Staubli VAL3: onF6Event.pgx

program onF6Event()
  local string l_sString
  local num l_nResult
  local bool l_bUndo
  local string l_sPaste
begin
  // look if the bButton is enable
  if bButton[5]
    //
    //  Duplicate
    //
    l_sPaste=sEvent
    call alreadyExist(l_sPaste,l_bUndo)
    if !l_bUndo
      call prog:duplicate(sEvent,l_sPaste,l_nResult)
      if l_nResult==0
        logMsg("[KERNEL] INTERFACE:Duplicate the program: "+sEvent+" to: "+l_sPaste)
        sEvent=l_sPaste
        call buildList()
      else
        popUpMsg("error code: "+toString("",l_nResult))
      endIf
    endIf
  endIf
end
